# EPICS alarm handler configuration: mps_database/bare/alarms/areas/mpln_l3b_mp04.alhConfig
GROUP NULL MPLN:L3B:MP04:1
$ALIAS MPS Link Node 70
$GUIDANCE
LTUH MPS
   Group Name: MPLN:L3B:MP04:1
   Summary PV:  MPLN:L3B:MP04:1:STATSUMY
$END
CHANNEL  MPLN:L3B:MP04:1    MPLN:L3B:MP04:1:MPS_EN_RBV		-----
CHANNEL  MPLN:L3B:MP04:1    MPLN:L3B:MP04:1:LC1_MODE_RBV		-----
